TYPE TTestResult :
STRUCT
    TestName         : T_MaxString;
    TestState        : T_MaxString;
    ImageRef         : T_MaxString;
    TestCompleteTime : T_MaxString;
END_STRUCT
END_TYPE

(* stored: Version 1.1.0.1, ProductVersion 3.1.4024.4
   DUT TTestResult: Id {ac11eadd-7f37-43d4-85bc-398c3d998e88} *)
